RoboDK station: Weld Script Graphical User Interface.rdk

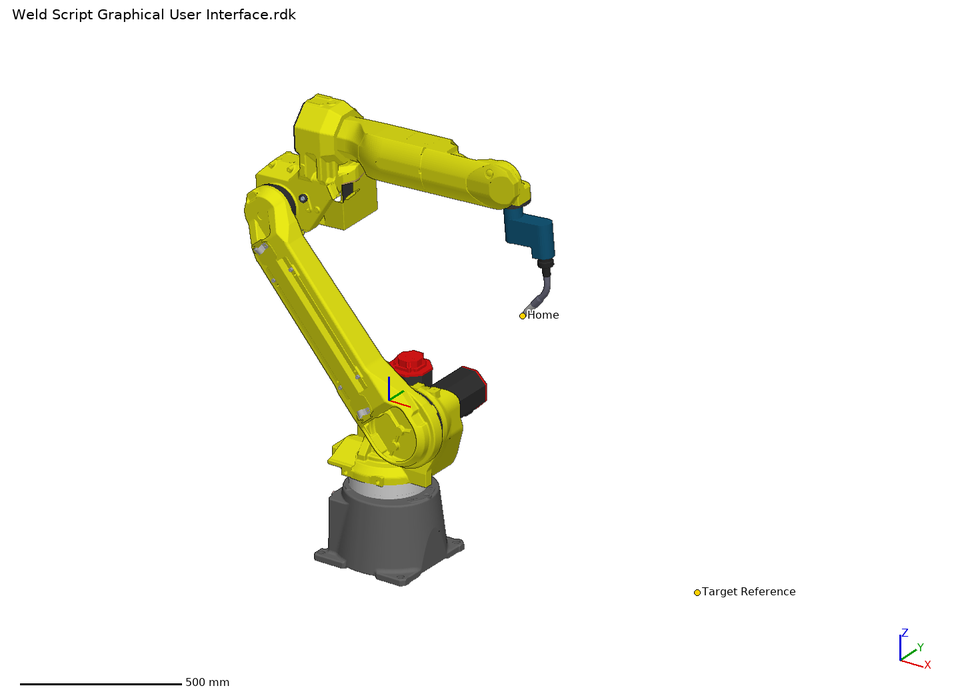
[picture v0: the station drawn from its stored meshes, robots at their saved joint values, targets as dots, program paths as lines]
Station Fanuc Sample GUI. Poses are relative to the parent item; angles as X-Y-Z fixed-axis rotations.
  - frame Fanuc ARC Mate 120iC Base at (0, 0, 0) mm
    - robot Fanuc ARC Mate 120iC: 6 axes, payload 3 kg, reach 1811 mm, repeatability 0.08 mm, weight 250 kg
        modified DH rows (alpha deg, a mm, theta deg, d mm): 0, 0, 0, 525; -90, 150, -90, 0; 0, 790, 0, 0; -90, 250, 0, 835; 90, 0, 0, 0; -90, 0, 0, 100
        base shift (0, 0, -525) mm
        joint limits [-185, -100, -345, -200, -140, -450] to [185, 160, 375.6, 200, 140, 450]; home [0, 0, 0, 0, 0, 0]; saved at [0, -40.164, 3.259, 0, -88.402, 180]
      - tool Weld gun, TCP at (-4, 0, 371.3) mm, rotated rx 0 ry 45 rz 0 deg, size 299.9 x 60 x 318.3 mm
    - target Home (joint target) at (503.79, 0, 431.51) mm, rotated rx -180 ry -40.14 rz 180 deg; joints [0, -40.164, 3.259, 0, -88.402, 180] of Fanuc ARC Mate 120iC
    - target Target Reference (Cartesian target) at (1163.72, 0, -334.69) mm, rotated rx -180 ry 0 rz -180 deg; joints [0, 17.951, -76.794, 0, 31.794, 180] of Fanuc ARC Mate 120iC
  - Python program Move Polygon GUI (listed below)

--- Python program Move Polygon GUI ---
# This example shows how RoboDK and the Python GUI tkinter can display graphical user interface to customize program generation according to certain parameters
# This example is an improvement of the weld Hexagon
from robolink import *    # API to communicate with RoboDK
from robodk import *      # robodk robotics toolbox
import threading

# Set up default parameters
PROGRAM_NAME = "DoWeld"     # Name of the program
APPROACH = 300              # Approach distance
RADIUS = 200                # Radius of the polygon
SPEED_WELD = 50             # Speed in mn/s of the welding path
SPEED_MOVE = 200            # Speed in mm/s of the approach/retract movements
SIDES = 8                   # Number of sides for the polygon
DRY_RUN = 1                 # If 0, it will generate SprayOn/SprayOff program calls, otherwise it will not activate the tool
RUN_MODE = RUNMODE_SIMULATE # Simulation behavior (simulate, generate program or generate the program and send it to the robot)
# use RUNMODE_SIMULATE to simulate only
# use RUNMODE_MAKE_ROBOTPROG to generate the program
# use RUNMODE_MAKE_ROBOTPROG_AND_UPLOAD to generate the program and send it to the robot


# Main program
def RunProgram():
    # Use default global variables
    global PROGRAM_NAME
    global APPROACH
    global RADIUS
    global SPEED_WELD
    global SPEED_MOVE
    global SIDES
    global DRY_RUN
    global RUN_MODE

    # Any interaction with RoboDK must be done through RDK:
    RDK = Robolink()

    # get the home target and the welding targets:
    home = RDK.Item('Home')
    target = RDK.Item('Target Reference')

    # get the robot as an item:
    robot = RDK.Item('', ITEM_TYPE_ROBOT)

    # impose the run mode
    RDK.setRunMode(RUN_MODE)
    # set the name of the generated program
    RDK.ProgramStart(PROGRAM_NAME, "", "", robot)

    # get the pose of the reference target (4x4 matrix representing position and orientation):
    poseref = target.Pose()

    # move the robot to home, then to an approach position
    robot.MoveJ(home)
    robot.setSpeed(SPEED_MOVE)
    robot.MoveJ(transl(0,0,APPROACH)*poseref)

    # make an polygon of n SIDES around the reference target
    for i in range(SIDES+1):
        ang = i*2*pi/SIDES #angle: 0, 60, 120, ...
        # Calculate next position
        posei = poseref*rotz(ang)*transl(RADIUS,0,0)*rotz(-ang)
        robot.MoveL(posei)

        # Impose weld speed only for the first point
        if i == 0:
            # Set weld speed and activate the gun after reaching the first point
            robot.setSpeed(SPEED_WELD)
            if not DRY_RUN:
                # Activate the spray right after we reached the first point
                robot.RunCodeCustom("SprayOn", INSTRUCTION_CALL_PROGRAM)

    # Stop the tool if we are not doing a dry run
    if not DRY_RUN:
        robot.RunCodeCustom("SprayOff", INSTRUCTION_CALL_PROGRAM)
    robot.setSpeed(SPEED_MOVE)

    # move back to the approach point, then home:
    robot.MoveL(transl(0,0,APPROACH)*poseref)
    robot.MoveJ(home)

    # Provoke program generation (automatic when RDK is finished)
    RDK.Finish()


# Use tkinter to display GUI menus
from tkinter import *

# Generate the main window
root = Tk()

# Use variables linked to the global variables
runmode = IntVar()
runmode.set(RUN_MODE)   # setting up default value

dryrun = IntVar()
dryrun.set(DRY_RUN)     # setting up default value

entry_name = StringVar()
entry_name.set(PROGRAM_NAME)

entry_speed = StringVar()
entry_speed.set(str(SPEED_WELD))

# Define feedback call
def ShowRunMode():
    print("Selected run mode: " + str(runmode.get()))

# Define a label and entry text for the program name
Label(root, text="Program name").pack()
Entry(root, textvariable=entry_name).pack()

# Define a label and entry text for the weld speed
Label(root, text="Weld speed (mm/s)").pack()
Entry(root, textvariable=entry_speed).pack()

# Define a check box to do a dry run
Checkbutton(root, text = "Dry run", variable=dryrun, onvalue=1, offvalue=0, height=5, width=20).pack()

# Add a display label for the run mode
Label(root, text="Run mode", justify=LEFT, padx=20).pack()

# Set up the run modes (radio buttons)
runmodes = [("Simulate",RUNMODE_SIMULATE),("Generate program",RUNMODE_MAKE_ROBOTPROG),("Send program to robot",RUNMODE_MAKE_ROBOTPROG_AND_START)]
for txt, val in runmodes:
    Radiobutton(root, text=txt, padx=20, variable=runmode, command=ShowRunMode, value=val).pack(anchor=W)

# Add a button and default action to execute the current choice of the user
def ExecuteChoice():
    def run_thread():
        global DRY_RUN
        global RUN_MODE
        global SPEED_WELD
        global PROGRAM_NAME
        DRY_RUN = dryrun.get()
        RUN_MODE = runmode.get()
        SPEED_WELD = float(entry_speed.get())
        PROGRAM_NAME = entry_name.get()
        # Run the main program once all the global variables have been set
        RunProgram()

    threading.Thread(target=run_thread).start()

Button(root, text='Simulate/Generate', command=ExecuteChoice).pack()

# Set window name
window_title = "Move Polygon Program"
root.title(window_title)

# We can embed the window into RoboDK as a docked window
# Make sure the window title is unique
EmbedWindow(window_title, size_w=200)

# Important to display the graphical user interface
root.mainloop()
